// TIA Portal V18 export
TYPE "LGasp_Tagliosega"
// stored: IsFailsafeCompliant false
   STRUCT
      nomeprogramma : WString[30];   // nome del programma trasferito dal PC
      Posizione : Struct   // asse traslazione, quota in mm
         inizialetaglio : LReal;
         intermedio1 : LReal;
         intermedio2 : LReal;
         intermedio3 : LReal;
         intermedio4 : LReal;
         intermedio5 : LReal;
         intermedio6 : LReal;
         finetaglio : LReal;
      END_STRUCT;
      Speedtraslazione : Struct   // asse traslazione, speed mm/min
         iniziale_intermedio1 : LReal;
         intermedio1_intermedio2 : LReal;
         intermedio2_intermedio3 : LReal;
         intermedio3_intermedio4 : LReal;
         intermedio4_intermedio5 : LReal;
         intermedio5_intermedio6 : LReal;
         intermedio6_fine : LReal;
         ritorno : LReal;
      END_STRUCT;
      Speedperiferica : Struct   // lama di taglio, speed periferica mm/min
         iniziale_intermedio1 : LReal;
         intermedio1_intermedio2 : LReal;
         intermedio2_intermedio3 : LReal;
         intermedio3_intermedio4 : LReal;
         intermedio4_intermedio5 : LReal;
         intermedio5_intermedio6 : LReal;
         intermedio6_fine : LReal;
         ritorno : LReal;
      END_STRUCT;
      Diametrolama : LReal;   // diametro reale lama in mm
      Tempociclotaglio : LReal;   // Durata taglio secondi (visualizzazione)
      Temporitorno : LReal;   // Durata ritorno lama secondi (visualizzazione)
      Posizionelama : LReal;   // Posizione asse traslazione lama mm (visualizzazione)
      Speedtraslaz : LReal;   // Velocità traslazione lama mm/min (visualizzazione)
      GiriLama : LReal;   // giri motore rotazione lama rpm (visualizzazione)
      Coppiatraslazione : LReal;   // coppia del motore traslazione lama (%)
      Coppiarotazione : LReal;   // coppia del motore rotazione lama (%)
      Limiti : Struct   // limiti dei valori inseribili nel PC impostati nel PLC
         pos_min : LReal := 0.0;   // limite minimo dei dati di posizione
         pos_max : LReal := 10000.0;   // limite massimo dei dati di posizione
         traslaz_min : LReal := 0.0;   // limite minimo dei dati di velocità traslazione
         traslaz_max : LReal := 10000.0;   // limite massimo dei dati di velocità traslazione
         ritorno_min : LReal := 0.0;   // limite minimo dei dati di velocità ritorno
         ritorno_max : LReal := 10000.0;   // limite massimo dei dati di velocità ritorno
         perif_min : LReal := 0.0;   // limite minimo dei dati di velocità periferica
         perif_max : LReal := 10000.0;   // limite massimo dei dati di velocità periferica
         diametro_min : LReal := 350.0;   // limite minimo diametro lama
         diametro_max : LReal := 450.0;   // limite massimo diametro lama
      END_STRUCT;
      Sensorotazione : Int;   // Visualizzazione su PC, 1=antiorario 2=orario
   END_STRUCT;
END_TYPE
